REGION Network 80: Check for Parameter Format Type
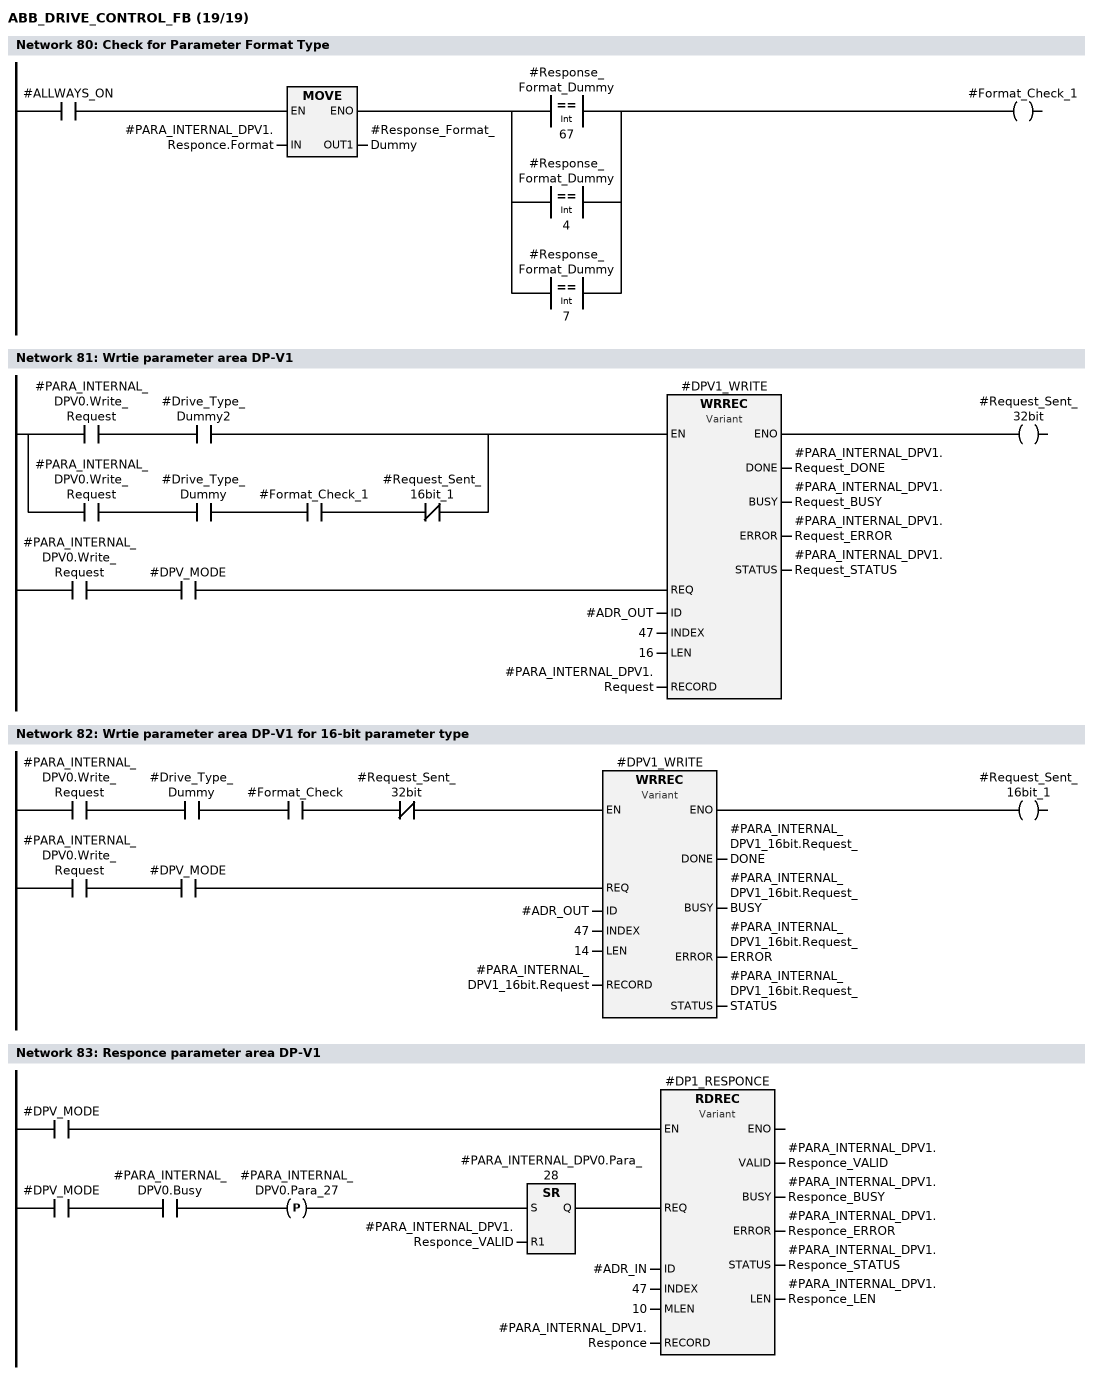
   RUNG wire#powerrail
      Contact( #ALLWAYS_ON )
      { S7_GenerateENO := "TRUE" } Move(in := #PARA_INTERNAL_DPV1.Responce.Format, out1 => #Response_Format_Dummy)
      wire#w1
      { S7_Templates := "SrcType := Int" } EQ_Contact(in1 := #Response_Format_Dummy, in2 := 67)
      wire#w2
      Coil( #Format_Check_1 )
   END_RUNG
   RUNG wire#w1
      { S7_Templates := "SrcType := Int" } EQ_Contact(in1 := #Response_Format_Dummy, in2 := 4)
   END_RUNG wire#w2
   RUNG wire#w1
      { S7_Templates := "SrcType := Int" } EQ_Contact(in1 := #Response_Format_Dummy, in2 := 7)
   END_RUNG wire#w2
   // the same network as SCL:
   // ENO of a box is taken as its EN; it also drops when the box reports an error
   IF #ALLWAYS_ON THEN #Response_Format_Dummy := #PARA_INTERNAL_DPV1.Responce.Format; END_IF;
   #Format_Check_1 := #ALLWAYS_ON AND ((#Response_Format_Dummy = 67) OR (#Response_Format_Dummy = 4) OR (#Response_Format_Dummy = 7));
END_REGION

REGION Network 81: Wrtie parameter area DP-V1
   RUNG wire#powerrail
      Contact( #PARA_INTERNAL_DPV0.Write_Request )
      Contact( #Drive_Type_Dummy2 )
      wire#w1
      { S7_Templates := "[ptr_type := Variant, id_type := HW_IO, index_type := DInt, len_type := UInt]" } #DPV1_WRITE.WRREC(REQ := wire#w2, ID := #ADR_OUT, INDEX := 47, LEN := 16, RECORD := #PARA_INTERNAL_DPV1.Request, DONE => #PARA_INTERNAL_DPV1.Request_DONE, BUSY => #PARA_INTERNAL_DPV1.Request_BUSY, ERROR => #PARA_INTERNAL_DPV1.Request_ERROR, STATUS => #PARA_INTERNAL_DPV1.Request_STATUS)
      Coil( #Request_Sent_32bit )
   END_RUNG
   RUNG wire#powerrail
      Contact( #PARA_INTERNAL_DPV0.Write_Request )
      Contact( #Drive_Type_Dummy )
      Contact( #Format_Check_1 )
      I_Contact( #Request_Sent_16bit_1 )
   END_RUNG wire#w1
   RUNG wire#powerrail
      Contact( #PARA_INTERNAL_DPV0.Write_Request )
      Contact( #DPV_MODE )
   END_RUNG wire#w2
   // the same network as SCL:
   #_w1 := (#PARA_INTERNAL_DPV0.Write_Request AND #Drive_Type_Dummy2) OR (#PARA_INTERNAL_DPV0.Write_Request AND #Drive_Type_Dummy AND #Format_Check_1 AND NOT #Request_Sent_16bit_1);
   #DPV1_WRITE(EN := #_w1,   // WRREC
               REQ := #PARA_INTERNAL_DPV0.Write_Request AND #DPV_MODE,
               ID := #ADR_OUT,
               INDEX := 47,
               LEN := 16,
               RECORD := #PARA_INTERNAL_DPV1.Request,
               DONE => #PARA_INTERNAL_DPV1.Request_DONE,
               BUSY => #PARA_INTERNAL_DPV1.Request_BUSY,
               ERROR => #PARA_INTERNAL_DPV1.Request_ERROR,
               STATUS => #PARA_INTERNAL_DPV1.Request_STATUS,
               ENO => #_w2);
   #Request_Sent_32bit := #_w2;
END_REGION

REGION Network 82: Wrtie parameter area DP-V1 for 16-bit parameter type
   RUNG wire#powerrail
      Contact( #PARA_INTERNAL_DPV0.Write_Request )
      Contact( #Drive_Type_Dummy )
      Contact( #Format_Check )
      I_Contact( #Request_Sent_32bit )
      { S7_Templates := "[ptr_type := Variant, id_type := HW_IO, index_type := DInt, len_type := UInt]" } #DPV1_WRITE.WRREC(REQ := wire#w1, ID := #ADR_OUT, INDEX := 47, LEN := 14, RECORD := #PARA_INTERNAL_DPV1_16bit.Request, DONE => #PARA_INTERNAL_DPV1_16bit.Request_DONE, BUSY => #PARA_INTERNAL_DPV1_16bit.Request_BUSY, ERROR => #PARA_INTERNAL_DPV1_16bit.Request_ERROR, STATUS => #PARA_INTERNAL_DPV1_16bit.Request_STATUS)
      Coil( #Request_Sent_16bit_1 )
   END_RUNG
   RUNG wire#powerrail
      Contact( #PARA_INTERNAL_DPV0.Write_Request )
      Contact( #DPV_MODE )
   END_RUNG wire#w1
   // the same network as SCL:
   #_w1 := #PARA_INTERNAL_DPV0.Write_Request AND #Drive_Type_Dummy AND #Format_Check AND NOT #Request_Sent_32bit;
   #DPV1_WRITE(EN := #_w1,   // WRREC
               REQ := #PARA_INTERNAL_DPV0.Write_Request AND #DPV_MODE,
               ID := #ADR_OUT,
               INDEX := 47,
               LEN := 14,
               RECORD := #PARA_INTERNAL_DPV1_16bit.Request,
               DONE => #PARA_INTERNAL_DPV1_16bit.Request_DONE,
               BUSY => #PARA_INTERNAL_DPV1_16bit.Request_BUSY,
               ERROR => #PARA_INTERNAL_DPV1_16bit.Request_ERROR,
               STATUS => #PARA_INTERNAL_DPV1_16bit.Request_STATUS,
               ENO => #_w2);
   #Request_Sent_16bit_1 := #_w2;
END_REGION

REGION Network 83: Responce parameter area DP-V1
   RUNG wire#powerrail
      Contact( #DPV_MODE )
      { S7_Templates := "[ptr_type := Variant, id_type := HW_IO, index_type := DInt, len_type := UInt]" } #DP1_RESPONCE.RDREC(REQ := wire#w1, ID := #ADR_IN, INDEX := 47, MLEN := 10, RECORD := #PARA_INTERNAL_DPV1.Responce, VALID => #PARA_INTERNAL_DPV1.Responce_VALID, BUSY => #PARA_INTERNAL_DPV1.Responce_BUSY, ERROR => #PARA_INTERNAL_DPV1.Responce_ERROR, STATUS => #PARA_INTERNAL_DPV1.Responce_STATUS, LEN => #PARA_INTERNAL_DPV1.Responce_LEN)
   END_RUNG
   RUNG wire#powerrail
      Contact( #DPV_MODE )
      Contact( #PARA_INTERNAL_DPV0.Busy )
      P_Trig( #PARA_INTERNAL_DPV0.Para_27 )
      S_SR(operand := #PARA_INTERNAL_DPV0.Para_28, r1 := #PARA_INTERNAL_DPV1.Responce_VALID)
   END_RUNG wire#w1
   // the same network as SCL:
   #_w1 := #DPV_MODE AND #PARA_INTERNAL_DPV0.Busy;
   #_w2 := #_w1 AND NOT #PARA_INTERNAL_DPV0.Para_27;   // rising edge
   #PARA_INTERNAL_DPV0.Para_27 := #_w1;
   IF #_w2 THEN
       #PARA_INTERNAL_DPV0.Para_28 := TRUE;   // SR flip-flop
   END_IF;
   IF #PARA_INTERNAL_DPV1.Responce_VALID THEN #PARA_INTERNAL_DPV0.Para_28 := FALSE; END_IF;
   IF #DPV_MODE THEN
       #DP1_RESPONCE(REQ := #PARA_INTERNAL_DPV0.Para_28,   // RDREC
                     ID := #ADR_IN,
                     INDEX := 47,
                     MLEN := 10,
                     RECORD := #PARA_INTERNAL_DPV1.Responce,
                     VALID => #PARA_INTERNAL_DPV1.Responce_VALID,
                     BUSY => #PARA_INTERNAL_DPV1.Responce_BUSY,
                     ERROR => #PARA_INTERNAL_DPV1.Responce_ERROR,
                     STATUS => #PARA_INTERNAL_DPV1.Responce_STATUS,
                     LEN => #PARA_INTERNAL_DPV1.Responce_LEN);
   END_IF;
END_REGION
END_FUNCTION_BLOCK
